// TIA Portal project "Project170625" (V17)

(* hardware
DEVICE "S7-1200 station_1"  S7-1200 Station
   slot 0: "Rack_0"  S7-1200 Rack  Rack  V1.0
   slot 1: "PLC_1"  CPU 1211C DC/DC/Rly  6ES7 211-1HE40-0XB0  V4.5
   slot 101: "CM 1241 (RS422/485)_1"  6ES7 241-1CH32-0XB0  V2.2
DEVICE "HMI_1"  KTP400 Comfort
   slot 0: "HMI_1"  KTP400 Comfort  6AV2 124-2DC01-0AX0  17.0.0.0
   slot 1: "HMI_RT_1"  KTP400 Comfort  6AV2 124-2DC01-0AX0  17.0.0.0
   slot 5: "HMI_1.IE_CP_1"  PROFINET Interface  17.0.0.0
      slot 1: "PROFINET Interface_1"  PROFINET Interface
         slot 1: "Port_1"  Port
   slot 7: "HMI_1.MPI/DP_CP_1"  MPI/DP Interface  17.0.0.0
*)

// ===== PLC "PLC_1"  CPU 1211C DC/DC/Rly =====

VAR_GLOBAL   // PLC tag table "Default tag table"
   "Clock_Byte" AT %MB0 : Byte;
   "Clock_10Hz" AT %M0.0 : Bool;
   "Clock_5Hz" AT %M0.1 : Bool;
   "Clock_2.5Hz" AT %M0.2 : Bool;
   "Clock_2Hz" AT %M0.3 : Bool;
   "Clock_1.25Hz" AT %M0.4 : Bool;
   "Clock_1Hz" AT %M0.5 : Bool;
   "Clock_0.625Hz" AT %M0.6 : Bool;
   "Clock_0.5Hz" AT %M0.7 : Bool;
   "System_Byte" AT %MB1 : Byte;
   "FirstScan" AT %M1.0 : Bool;
   "DiagStatusUpdate" AT %M1.1 : Bool;
   "AlwaysTRUE" AT %M1.2 : Bool;
   "AlwaysFALSE" AT %M1.3 : Bool;
   "Capteur A" AT %M30.0 : Bool;
   "Capteur B" AT %M30.1 : Bool;
   "Capteur C" AT %M30.2 : Bool;
   "Etape 1" AT %M70.0 : Bool;
   "Etape 2" AT %M70.1 : Bool;
   "Etape 3" AT %M70.2 : Bool;
   "Etape 4" AT %M70.3 : Bool;
   "Etape 5" AT %M70.4 : Bool;
   "Droite" AT %Q0.0 : Bool;
   "Gauche" AT %Q0.1 : Bool;
   "DCY" AT %I0.1 : Bool;
   "Tag_1" AT %M20.0 : Bool;
   "Tag_2" AT %M20.1 : Bool;
   "Deplacement" AT %MW10 : Int;
   "TRANSFERT" AT %M60.0 : Bool;
   "COMPTEUR" AT %MW100 : Int;
END_VAR

// folder: System blocks/Program resources

DATA_BLOCK "IEC_Timer_0_DB"   // DB1
{ S7_Optimized_Access := 'TRUE' }
AUTHOR : Simatic
FAMILY : IEC
NAME : IEC_TMR
VERSION : 1.0
// stored: InstanceOfName IEC_TIMER
"IEC_TIMER"
BEGIN
END_DATA_BLOCK

DATA_BLOCK "IEC_Timer_0_DB_1"   // DB2
{ S7_Optimized_Access := 'TRUE' }
AUTHOR : Simatic
FAMILY : IEC
NAME : IEC_TMR
VERSION : 1.0
// stored: InstanceOfName IEC_TIMER
"IEC_TIMER"
BEGIN
END_DATA_BLOCK

DATA_BLOCK "IEC_Timer_0_DB_2"   // DB3
{ S7_Optimized_Access := 'TRUE' }
AUTHOR : Simatic
FAMILY : IEC
NAME : IEC_TMR
VERSION : 1.0
// stored: InstanceOfName IEC_TIMER
"IEC_TIMER"
BEGIN
END_DATA_BLOCK

DATA_BLOCK "IEC_Timer_0_DB_3"   // DB4
{ S7_Optimized_Access := 'TRUE' }
AUTHOR : Simatic
FAMILY : IEC
NAME : IEC_TMR
VERSION : 1.0
// stored: InstanceOfName IEC_TIMER
"IEC_TIMER"
BEGIN
END_DATA_BLOCK

DATA_BLOCK "IEC_Counter_0_DB"   // DB6
{ S7_Optimized_Access := 'TRUE' }
AUTHOR : Simatic
FAMILY : IEC
NAME : CNTR
VERSION : 1.0
// stored: InstanceOfName IEC_COUNTER
"IEC_COUNTER"
BEGIN
END_DATA_BLOCK

// folder: (top level)

FUNCTION "TEST" : Void   // FC1, LAD
{ S7_Optimized_Access := 'TRUE' }
VERSION : 0.1
   VAR_TEMP   // added for the SCL form of the ladder/FBD networks
      _w1 : Bool;
   END_VAR
BEGIN

REGION Network 1
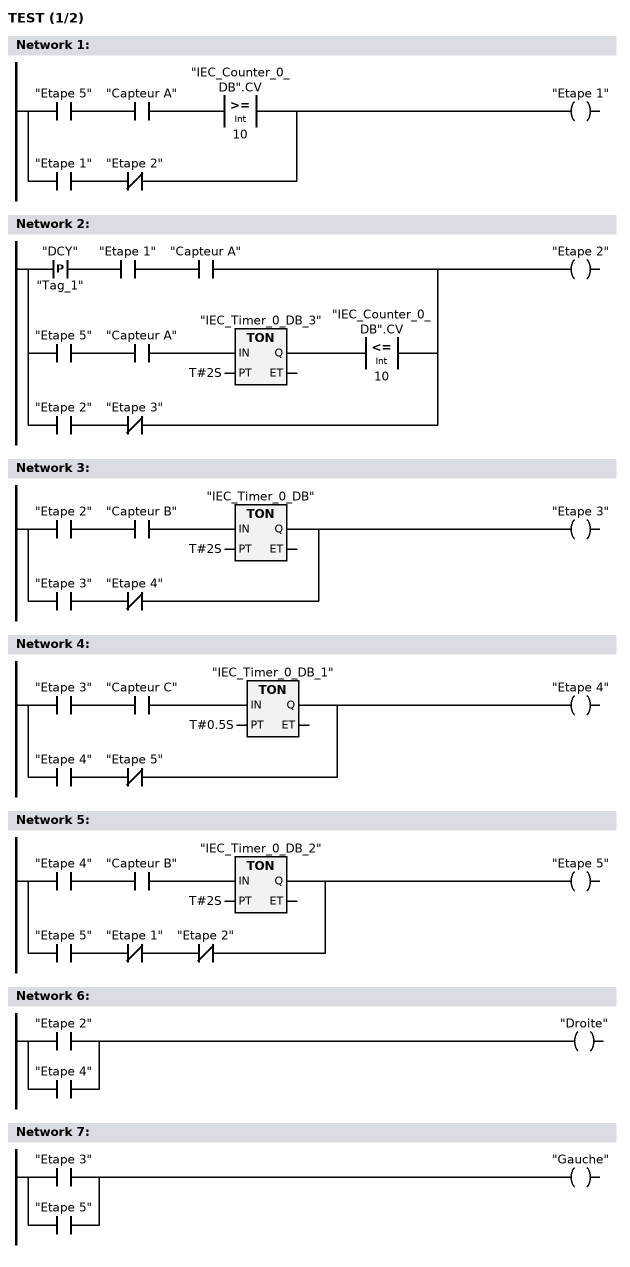
   RUNG wire#powerrail
      Contact( "Etape 5" )
      Contact( "Capteur A" )
      { S7_Templates := "SrcType := Int" } GE_Contact(in1 := "IEC_Counter_0_DB".CV, in2 := 10)
      wire#w1
      Coil( "Etape 1" )
   END_RUNG
   RUNG wire#powerrail
      Contact( "Etape 1" )
      I_Contact( "Etape 2" )
   END_RUNG wire#w1
   // the same network as SCL:
   "Etape 1" := ("Etape 5" AND "Capteur A" AND ("IEC_Counter_0_DB".CV >= 10)) OR ("Etape 1" AND NOT "Etape 2");
END_REGION

REGION Network 2
   #_w1 := "DCY" AND NOT "Tag_1";   // rising edge of "DCY"
   "Tag_1" := "DCY";
   "IEC_Timer_0_DB_3".TON(IN := "Etape 5" AND "Capteur A", PT := T#2S);
   "Etape 2" := (#_w1 AND "Etape 1" AND "Capteur A") OR ("IEC_Timer_0_DB_3".Q AND ("IEC_Counter_0_DB".CV <= 10)) OR ("Etape 2" AND NOT "Etape 3");
END_REGION

REGION Network 3
   "IEC_Timer_0_DB".TON(IN := "Etape 2" AND "Capteur B", PT := T#2S);
   "Etape 3" := "IEC_Timer_0_DB".Q OR ("Etape 3" AND NOT "Etape 4");
END_REGION

REGION Network 4
   "IEC_Timer_0_DB_1".TON(IN := "Etape 3" AND "Capteur C", PT := T#0.5S);
   "Etape 4" := "IEC_Timer_0_DB_1".Q OR ("Etape 4" AND NOT "Etape 5");
END_REGION

REGION Network 5
   "IEC_Timer_0_DB_2".TON(IN := "Etape 4" AND "Capteur B", PT := T#2S);
   "Etape 5" := "IEC_Timer_0_DB_2".Q OR ("Etape 5" AND NOT "Etape 1" AND NOT "Etape 2");
END_REGION

REGION Network 6
   RUNG wire#powerrail
      Contact( "Etape 2" )
      wire#w1
      Coil( "Droite" )
   END_RUNG
   RUNG wire#powerrail
      Contact( "Etape 4" )
   END_RUNG wire#w1
   // the same network as SCL:
   "Droite" := "Etape 2" OR "Etape 4";
END_REGION

REGION Network 7
   RUNG wire#powerrail
      Contact( "Etape 3" )
      wire#w1
      Coil( "Gauche" )
   END_RUNG
   RUNG wire#powerrail
      Contact( "Etape 5" )
   END_RUNG wire#w1
   // the same network as SCL:
   "Gauche" := "Etape 3" OR "Etape 5";
END_REGION

REGION Network 8
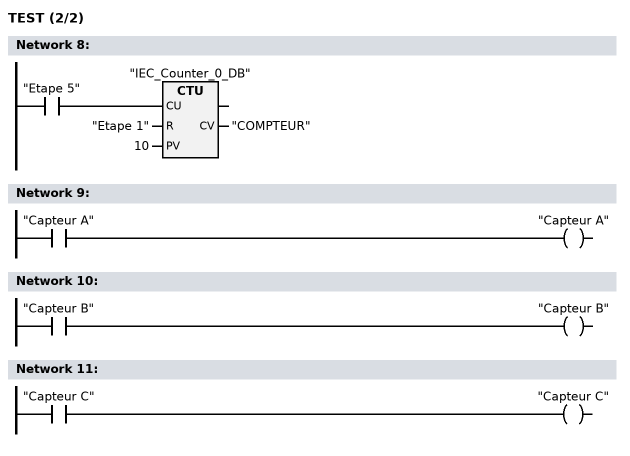
   "IEC_Counter_0_DB".CTU(CU := "Etape 5", R := "Etape 1", PV := 10, CV => "COMPTEUR");
END_REGION

REGION Network 9
   RUNG wire#powerrail
      Contact( "Capteur A" )
      Coil( "Capteur A" )
   END_RUNG
   // the same network as SCL:
   "Capteur A" := "Capteur A";
END_REGION

REGION Network 10
   RUNG wire#powerrail
      Contact( "Capteur B" )
      Coil( "Capteur B" )
   END_RUNG
   // the same network as SCL:
   "Capteur B" := "Capteur B";
END_REGION

REGION Network 11
   RUNG wire#powerrail
      Contact( "Capteur C" )
      Coil( "Capteur C" )
   END_RUNG
   // the same network as SCL:
   "Capteur C" := "Capteur C";
END_REGION
END_FUNCTION

FUNCTION "Block_1" : Void   // FC2, LAD
{ S7_Optimized_Access := 'TRUE' }
VERSION : 0.1
BEGIN

REGION Network 1
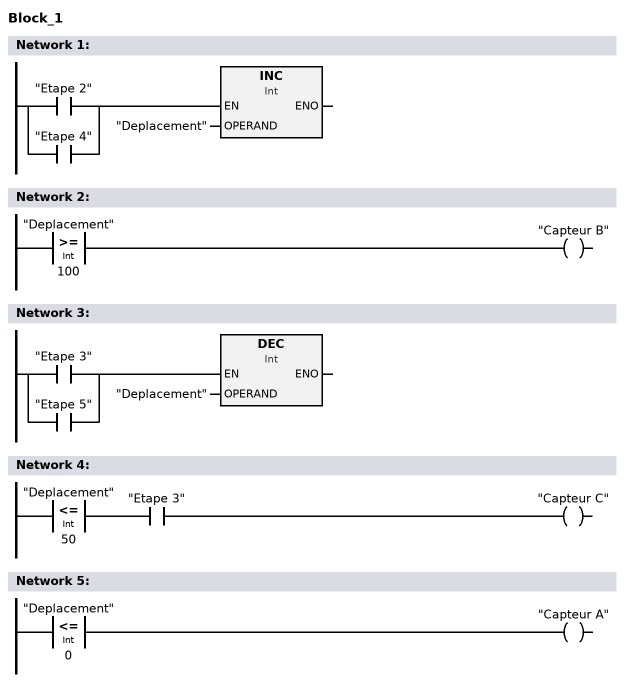
   RUNG wire#powerrail
      Contact( "Etape 2" )
      wire#w1
      { S7_Templates := "DestType := Int" } Inc( "Deplacement" )
   END_RUNG
   RUNG wire#powerrail
      Contact( "Etape 4" )
   END_RUNG wire#w1
   // the same network as SCL:
   IF "Etape 2" OR "Etape 4" THEN "Deplacement" := "Deplacement" + 1; END_IF;
END_REGION

REGION Network 2
   RUNG wire#powerrail
      { S7_Templates := "SrcType := Int" } GE_Contact(in1 := "Deplacement", in2 := 100)
      Coil( "Capteur B" )
   END_RUNG
   // the same network as SCL:
   "Capteur B" := "Deplacement" >= 100;
END_REGION

REGION Network 3
   RUNG wire#powerrail
      Contact( "Etape 3" )
      wire#w1
      { S7_Templates := "DestType := Int" } Dec( "Deplacement" )
   END_RUNG
   RUNG wire#powerrail
      Contact( "Etape 5" )
   END_RUNG wire#w1
   // the same network as SCL:
   IF "Etape 3" OR "Etape 5" THEN "Deplacement" := "Deplacement" - 1; END_IF;
END_REGION

REGION Network 4
   RUNG wire#powerrail
      { S7_Templates := "SrcType := Int" } LE_Contact(in1 := "Deplacement", in2 := 50)
      Contact( "Etape 3" )
      Coil( "Capteur C" )
   END_RUNG
   // the same network as SCL:
   "Capteur C" := ("Deplacement" <= 50) AND "Etape 3";
END_REGION

REGION Network 5
   RUNG wire#powerrail
      { S7_Templates := "SrcType := Int" } LE_Contact(in1 := "Deplacement", in2 := 0)
      Coil( "Capteur A" )
   END_RUNG
   // the same network as SCL:
   "Capteur A" := "Deplacement" <= 0;
END_REGION
END_FUNCTION

ORGANIZATION_BLOCK "Main"   // OB1, LAD, ProgramCycle
TITLE = "Main Program Sweep (Cycle)"
{ S7_Optimized_Access := 'TRUE' }
VERSION : 0.1
   VAR_INPUT
      Initial_Call : Bool;   // Initial call of this OB
      Remanence : Bool;   // =True, if remanent data are available
   END_VAR
BEGIN

REGION Network 1
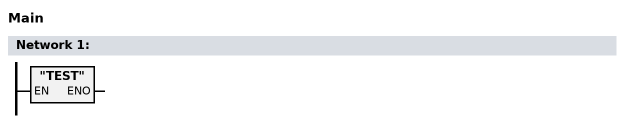
   RUNG wire#powerrail
      "TEST"()
   END_RUNG
   // the same network as SCL:
   "TEST"();
END_REGION
END_ORGANIZATION_BLOCK

ORGANIZATION_BLOCK "Cyclic interrupt_1"   // OB31, LAD, CyclicInterrupt
{ S7_Optimized_Access := 'TRUE' }
VERSION : 0.1
   VAR_INPUT
      Initial_Call : Bool;   // Initial call of this OB
      Event_Count : Int;   // Events discarded
   END_VAR
BEGIN

REGION Network 1
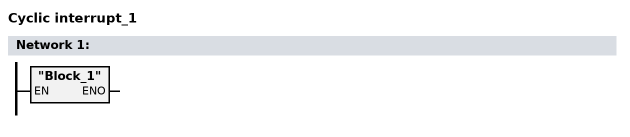
   RUNG wire#powerrail
      "Block_1"()
   END_RUNG
   // the same network as SCL:
   "Block_1"();
END_REGION
END_ORGANIZATION_BLOCK

ORGANIZATION_BLOCK "Startup"   // OB100, LAD, Startup
TITLE = "Complete Restart"
{ S7_Optimized_Access := 'TRUE' }
VERSION : 0.1
   VAR_INPUT
      LostRetentive : Bool;   // True if retentive data are lost
      LostRTC : Bool;   // True if date and time are lost
   END_VAR
BEGIN

REGION Network 1
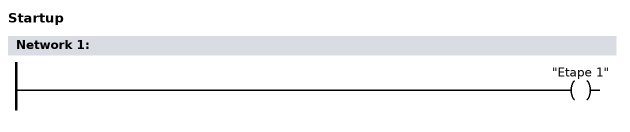
   RUNG wire#powerrail
      Coil( "Etape 1" )
   END_RUNG
   // the same network as SCL:
   "Etape 1" := TRUE;
END_REGION
END_ORGANIZATION_BLOCK

(* ===== HMI "HMI_RT_1" =====
system functions are stored by id; their names below are inferred from use
connection "HMI_Connection_1": ETHERNET, S7_1200_OMS

HMI tags "Default tag table"
   "HMI_Tag_1" : Bool = PLC DCY AT %I0.1, 1 s
   "Gauche" : Bool = PLC Gauche AT %Q0.1, 1 s
   "Droite" : Bool = PLC Droite AT %Q0.0, 1 s
   "Deplacement" : Int = PLC Deplacement AT %MW10, 1 s
   "Capteur A" : Bool = PLC "Capteur A" AT %M30.0, 1 s
   "Capteur C" : Bool = PLC "Capteur C" AT %M30.2, 1 s
   "Capteur B" : Bool = PLC "Capteur B" AT %M30.1, 1 s
   "COMPTEUR" : Int = PLC COMPTEUR AT %MW100, 1 s

Template "Template_1" 480x272
   Button "Exit" at 379,208 size 63x63; TextOff 'Exit'; PictureOff "ExitRuntime_KTP400_Comfort_TR"; PictureOn "ExitRuntime_KTP400_Comfort_TR"
      on Release: StopRuntime(0)
   Button "Language" at 265,208 size 63x63; TextOff 'Language'; PictureOff "ToggleLanguage_KTP400_Comfort_TR"; PictureOn "ToggleLanguage_KTP400_Comfort_TR"
      on Release: function_fb9197e8(-1)
   Button "Log on" at 151,208 size 63x63; TextOff 'Log on'; PictureOff "Login_KTP400_Comfort_TR"; PictureOn "Login_KTP400_Comfort_TR"
      on Release: function_a2a04561()
   Button "Start screen" at 37,208 size 63x63; TextOff 'Start screen'; PictureOff "NavigateHome_KTP400_Comfort_TR"; PictureOn "NavigateHome_KTP400_Comfort_TR"
      on Release: ActivateScreen("Accueil", 0)
   AlarmView "Alarm view_Unacknowledged" at 0,0 size 480x18

screen "Accueil" 480x272, template "Template_1"
   Softkey "Softkey_F1" at 0,0 size 0x0
      on KeyDown: ActivateScreen("Accueil", 0)
   Button "Button_1" at 5,155 size 97x36; TextOff 'DCY'
      on Press: InvertBit("HMI_Tag_1")
   DateTimeField "Date/time field_1" at 0,0 size 202x29
   Softkey "Softkey_F2" at 0,0 size 0x0
      on KeyDown: ActivateScreen("Screen_1", 0)
   Softkey "Softkey_F3" at 0,0 size 0x0
      on KeyDown: ActivateScreen("Screen_2", 0)

screen "Screen_1" 480x272
   Circle "Circle_1" at 48,94 size 63x63
      Appearance <- "Gauche"
   Circle "Circle_2" at 359,93 size 63x63
      Appearance <- "Droite"
   TextField "Text field_1" at 66,106 size 26x37; Text 'G'
   TextField "Text field_2" at 378,106 size 26x37; Text 'D'
   Softkey "Softkey_F2" at 0,0 size 0x0
      on KeyDown: ActivateScreen("Screen_1", 0)
   Softkey "Softkey_F1" at 0,0 size 0x0
      on KeyDown: ActivateScreen("Accueil", 0)
   Softkey "Softkey_F3" at 0,0 size 0x0
      on KeyDown: ActivateScreen("Screen_2", 0)

screen "Screen_2" 480x272
   Softkey "Softkey_F3" at 0,0 size 0x0
      on KeyDown: ActivateScreen("Screen_2", 0)
   Group "Group" at 0,103 size 84x62
      HorizontalMovement <- "Deplacement"
   Circle "Circle_3" at 218,164 size 44x44
      Appearance <- "Capteur C"
   Circle "Circle_4" at 19,168 size 44x44
      Appearance <- "Capteur A"
   Circle "Circle_5" at 415,165 size 44x44
      Appearance <- "Capteur B"
   TextField "Text field_1" at 28,165 size 28x43; Text 'A'
   TextField "Text field_2" at 423,162 size 28x43; Text 'B'
   TextField "Text field_3" at 225,162 size 27x43; Text 'C'
   IOField "I/O field_1" at 19,5 size 96x32; FormatPattern s99999
      ProcessValue <- "Deplacement"
   IOField "I/O field_2" at 356,6 size 96x32; FormatPattern s99999
      ProcessValue <- "COMPTEUR"
   Softkey "Softkey_F1" at 0,0 size 0x0
      on KeyDown: ActivateScreen("Accueil", 0)
   Softkey "Softkey_F2" at 0,0 size 0x0
      on KeyDown: ActivateScreen("Screen_1", 0)
*)